(* PLC project ActionMemberFixture *)

PROGRAM PLC_TEST

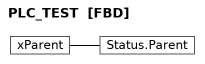
(* FBD diagram, written out as Structured Text *)
Status.Parent := xParent;

ACTION ACT_TEST:
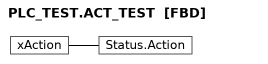
(* FBD diagram, written out as Structured Text *)
Status.Action := xAction;
END_ACTION
END_PROGRAM
